(*
SPDX-FileCopyrightText: © 2026 Oleksandr Tiutyk <trofimich@gmail.com>
SPDX-License-Identifier: MIT
License: https://opensource.org/license/mit
*)

(*!
<summary>
Beckhoff EL1809: 16-channel HD digital input terminal (24 V DC, 3 ms filter).
</summary>
<description>
Process image mapping structure for the high-density EL1809 EtherCAT terminal with 16 discrete 24 V DC inputs.
When used for I/O, link located fields or their containing buffers to the matching selected PDOs.
The record is not a packed wire buffer; compiler padding is not part of the device specification.
Unlinked/default values do not prove valid I/O. The caller evaluates bus/channel validity before use.
Use one owner task per instance and externally synchronize other access; multi-field snapshots are not atomic.
Copies store data without creating hardware links. Keep borrowed field references valid while consumers are bound.
This passive record performs no validation, synchronization, configuration or protocol advancement.
</description>
*)
TYPE EL1809 :
STRUCT
	Ch01 AT %I* : BOOL;
	Ch02 AT %I* : BOOL;
	Ch03 AT %I* : BOOL;
	Ch04 AT %I* : BOOL;
	Ch05 AT %I* : BOOL;
	Ch06 AT %I* : BOOL;
	Ch07 AT %I* : BOOL;
	Ch08 AT %I* : BOOL;
	Ch09 AT %I* : BOOL;
	Ch10 AT %I* : BOOL;
	Ch11 AT %I* : BOOL;
	Ch12 AT %I* : BOOL;
	Ch13 AT %I* : BOOL;
	Ch14 AT %I* : BOOL;
	Ch15 AT %I* : BOOL;
	Ch16 AT %I* : BOOL;	
END_STRUCT
END_TYPE

(* stored: Version 1.1.0.1, ProductVersion 3.1.4026.20
   DUT EL1809: Id {8fe0bc1e-6d21-40c6-9d20-61b703115a67} *)
